Universal Robots PolyScope program: orange_Triangle.urp

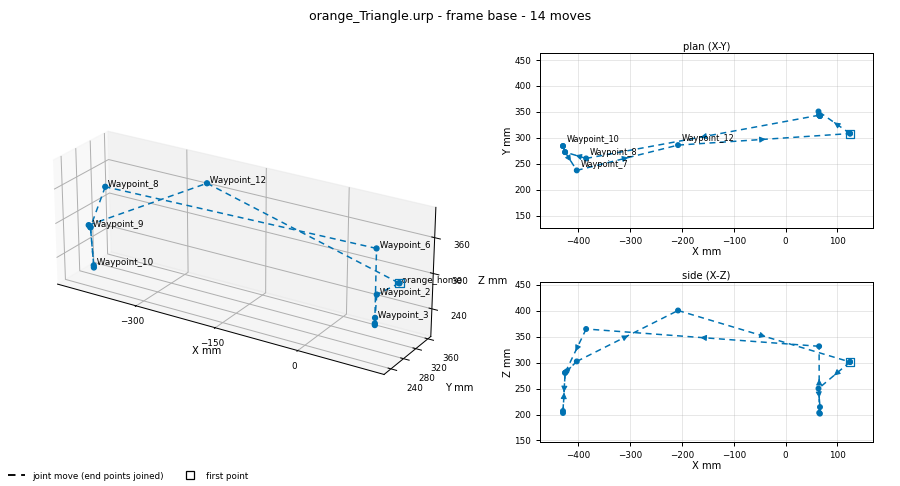
[picture p0: tool path of orange_Triangle.urp in frame base, 14 of 14 moves have a stored position in this frame; points joined in program order, loops and branches not executed]
Program orange_Triangle (installation=default directory=/programs/usbdisk/Zahra1/orangi createdIn=5.11.11.1010533 lastSavedIn=5.11.11.1010533 robotSerialNumber=20205300864)
Calibrated DH parameters: a=[-0.000166, -0.243494, -0.153108, 0.000057, -0.000123, 0]; d=[0.151897, -1.34267, 53.988124, -52.514559, 0.085283, 0.092193]; alpha=[1.572472, -0.003756, 0.002824, 1.570807, -1.572621, 0]; deltaTheta=[0, 0.020704, 7.033215, -0.770746, 0.000004, 0]
Robot Program (runOnlyOnce=true)
  MoveJ speed 60 deg/s, acceleration 80 deg/s^2 (useActiveTCP=true) feature=Base
    Waypoint orange_home: TCP in base x=124.286 y=308.277 z=301.462 mm, rx=2.2499 ry=-2.1846 rz=-0.0963 rad; joints [-269.66, -91.226, -90.279, -86.086, 92.69, 808.818] deg
    Waypoint Waypoint_2: TCP in base x=63.449 y=350.84 z=250.212 mm, rx=2.1934 ry=-2.2182 rz=0.0229 rad; joints [-258.977, -99.711, -93.213, -78.37, 90.598, 821.791] deg
    Waypoint Waypoint_3: TCP in base x=66.327 y=341.927 z=214.475 mm, rx=-2.2737 ry=2.1642 rz=0.0302 rad; joints [-259.174, -99.799, -104.247, -64.87, 90.549, 818.163] deg
    Waypoint Waypoint_4: TCP in base x=66.166 y=342.119 z=201.786 mm, rx=-2.2737 ry=2.1643 rz=0.0301 rad; joints [-259.157, -101.18, -106.327, -61.411, 90.548, 818.191] deg
    URCap Gripper (Robotiq_Grippers, Robotiq Inc.) dataModel(position=70.98039215686275, force=97.0, speed=52.0, positionInDouble=70.98039215686275, forceInDouble=97.0, speedInDouble=52.0, slaveIds=[9], blocking=true, robotCompliant=false)
    Waypoint Waypoint_5: TCP in base x=64.862 y=344.322 z=203.4 mm, rx=-2.2328 ry=2.2031 rz=0.0039 rad; joints [-258.811, -101.48, -105.144, -62.999, 89.868, 820.583] deg
    Waypoint Waypoint_6: TCP in base x=64.646 y=343.651 z=331.71 mm, rx=-2.2328 ry=2.2031 rz=0.0037 rad; joints [-258.694, -96.408, -75.672, -97.55, 89.83, 820.626] deg
    Waypoint Waypoint_8: TCP in base x=-384.713 y=260.289 z=365.043 mm, rx=-2.7605 ry=1.4193 rz=0.3055 rad; joints [-197.007, -129.248, -23.084, -106.715, 86.571, 847.08] deg
    Waypoint Waypoint_9: TCP in base x=-425.297 y=272.448 z=280.636 mm, rx=-2.7568 ry=1.4118 rz=0.1463 rad; joints [-196.994, -140.774, -23.087, -101.113, 86.57, 847.08] deg
    Waypoint Waypoint_10: motionParameters(jointSpeed=0.698132 jointAcceleration=0.349066 cartesianSpeed=0.25 cartesianAcceleration=1.2); TCP in base x=-429.415 y=284.093 z=206.849 mm, rx=-2.7217 ry=1.5556 rz=0.0366 rad; joints [-198.665, -144.072, -35.256, -89.324, 89.226, 850.841] deg
    Waypoint Waypoint_1: TCP in base x=-429.334 y=284.239 z=203.087 mm, rx=-2.7198 ry=1.5539 rz=0.0353 rad; joints [-198.663, -144.099, -36.186, -88.443, 89.097, 850.826] deg
    URCap Gripper (Robotiq_Grippers, Robotiq Inc.) dataModel(position=40.3921568627451, force=97.0, speed=52.0, positionInDouble=40.3921568627451, forceInDouble=97.0, speedInDouble=52.0, slaveIds=[9], blocking=true, robotCompliant=false)
    Waypoint Waypoint_9: TCP in base x=-425.297 y=272.448 z=280.636 mm, rx=-2.7568 ry=1.4118 rz=0.1463 rad; joints [-196.994, -140.774, -23.087, -101.113, 86.57, 847.08] deg
    Waypoint Waypoint_7: TCP in base x=-402.796 y=237.199 z=302.521 mm, rx=-2.8876 ry=0.7416 rz=0.258 rad; joints [-192.443, -123.065, -50.995, -86.186, 81.04, 825.641] deg
    Waypoint Waypoint_12: TCP in base x=-207.468 y=285.965 z=400.743 mm, rx=-2.8284 ry=1.1349 rz=-0.0569 rad; joints [-210.714, -103.223, -47.171, -120.801, 84.288, 823.123] deg
    Waypoint orange_home: TCP in base x=124.286 y=308.277 z=301.462 mm, rx=2.2499 ry=-2.1846 rz=-0.0963 rad; joints [-269.66, -91.226, -90.279, -86.086, 92.69, 808.818] deg
